// TIA Portal V17 export
// export: Created 2024-03-30T11:14:56.0079882Z, ExportSetting WithDefaults, DisplayName Totally Integrated Automation Portal, DisplayVersion V17, DisplayName TIA Portal Openness, DisplayVersion V17, DisplayName TIA Portal Version Control Interface, DisplayVersion V17, DisplayName STEP 7 Professional, DisplayVersion V17, DisplayName STEP 7 Safety, DisplayVersion V17, DisplayName WinCC Advanced, DisplayVersion V17
TYPE "typ_MQTT_Interface_Dashboard"
// stored: IsFailsafeCompliant false
   STRUCT
      Subscribe : "typ_MQTT_Interface_Dashboard_Subscribe";
      Publish { S7_SetPoint := 'True'} : "typ_MQTT_ Interface_Dashboard_Publish";
   END_STRUCT;
END_TYPE
